{attribute 'qualified_only'}
{attribute 'strict'}
{attribute 'to_string'}
TYPE E_SeqDoorLock :
(
	INIT := 0,
	LOCKED,
	ACCESS_REQUEST_PENDING,
	UNLOCKED,
	DOOR_CLOSED,
	DOOR_OPENED,
	ERROR
);
END_TYPE

(* stored: Version 1.1.0.1, ProductVersion 3.1.4024.12
   DUT E_SeqDoorLock: Id {6e07db46-519a-4368-a773-15c4098f34fa} *)
